INTERFACE I_FSM

METHOD Event
VAR_INPUT
	e : INT;
END_VAR
END_METHOD

END_INTERFACE

(* stored: Version 1.1.0.1, ProductVersion 3.1.4024.12
   Itf I_FSM: Id {4e01c3db-1ac2-03ab-2dbe-1551dcfb6cab}
   Method Event: Id {1c98c286-66af-04ea-2402-d61edcdfeaa5} *)
